FUNCTION_BLOCK PUBLIC FB_Button
VAR_INPUT
	ProcessFinished : BOOL;
END_VAR

VAR
	ButtonInput AT%I* : BOOL;
	ButtonLight AT%Q* : BOOL := TRUE;
	Click : F_TRIG;
	fbTon : TON := (PT :=T#0.3S); 
	state : INT := 0;
END_VAR

VAR_OUTPUT
	bMotorOn : BOOL;
	FlipProcess : BOOL; 
END_VAR

CASE state OF
	
	0:
		Click(CLK := ButtonInput);
		IF Click.Q THEN
			state := 20;
			FlipProcess := FALSE;
		END_IF
		fbTon(IN := TRUE);
		IF fbTON.Q THEN
			fbTON(IN := FALSE);	
			ButtonLight := FALSE;
			state := 10;
		END_IF
		bMotorOn := FALSE;
		
	10:
		Click(CLK := ButtonInput);
		IF Click.Q THEN
			state := 20;
			FlipProcess := FALSE;
		END_IF
		fbTon(IN := TRUE);
		IF fbTON.Q THEN
			fbTON(IN := FALSE);	
			ButtonLight := TRUE;
			state := 0;
		END_IF
		bMotorOn := FALSE;
		
	20: 
		Click(CLK := ButtonInput);
		IF Click.Q  OR ProcessFinished THEN
			state := 0;
		END_IF
		ButtonLight := TRUE;	
		bMotorOn := TRUE;
	
END_CASE

END_FUNCTION_BLOCK

(* stored: Version 1.1.0.1, ProductVersion 3.1.4024.12
   POU FB_Button: Id {c88f4204-26c4-45d9-b1c4-17a86b7fe003}, SpecialFunc None *)
